(* IEC 61131-3 sources: LANTA/1.8QVPLC1.0/phase-calibration/codex-manual-v2-20260911, 4 files *)

(* ---- GVL_PhaseCal.st ---- *)
{attribute 'qualified_only'}
VAR_GLOBAL
    (* Commands: non-retained. Never FORCE these or axis commands. *)
    xStart : BOOL;
    xAbort : BOOL;
    xReset : BOOL;
    (* Commissioning interlock: confirm aligned reads with the actual protocol first.
       recSize>=16 alone is NOT a frame/header/checksum verification. *)
    xRxAlignmentConfirmed : BOOL := FALSE;
    lrCurrentPhaseDeg : LREAL := 0;
    iPhaseDirection : INT := 0; (* unknown=0, CCW=+1, CW=-1 *)
    (* Manual configuration. HPBW is the FULL -3 dB width in degrees. *)
    lrBeamAzDeg : LREAL := 0; (* required *)
    lrBeamElDeg : LREAL := 0; (* required *)
    lrScanFraction : LREAL := 0.2;
    lrTargetVolt : LREAL := 1.0; (* at 0.2 HPBW, independent of scan fraction *)
    lrCurrentGainAz : LREAL := 1;
    lrCurrentGainEl : LREAL := 1;
    iGainUnit : INT := 0; (* 0=linear voltage multiplier; 1=20*log10 multiplier dB *)
    iGainOrder : INT := 0; (* required: 1=gains before common rotation; 2=after *)
    lrGainMin : LREAL := 0.01; (* limits in selected device gain units *)
    lrGainMax : LREAL := 100;
    lrLegTimeSec : LREAL := 1.1;
    lrSettleSec : LREAL := 0.6; (* total dwell, including delay/settling and collection *)
    lrRxDelaySec : LREAL := 0.15; (* measured upper bound of receiver/filter delay *)
    lrStableSec : LREAL := 0.10;
    lrSampleIntervalSec : LREAL := 0.02;
    lrPositionToleranceDeg : LREAL := 0.002; (* mechanical per-axis *)
    lrMaxAxisOffsetDeg : LREAL := 0.1; (* commissioning ceiling; explicitly review if changed *)
    lrMaxVelocityDegSec : LREAL := 0; (* required mechanical per-axis limit *)
    lrMaxAccelerationDegSec2 : LREAL := 0; (* required mechanical per-axis limit *)
    lrMinCosEl : LREAL := 0.1; (* reject near zenith *)
    lrMaxOrthErrorDeg : LREAL := 3;
    lrMinEbN0 : LREAL := 29; (* legacy compatibility; no new EbN0 gate *)

    xGainValid : BOOL;
    lrGainFactorAz, lrGainFactorEl : LREAL;
    lrSuggestedGainAz, lrSuggestedGainEl : LREAL;
    lrSensitivityAz, lrSensitivityEl : LREAL; (* V/degree after proposed rotation, before new gain *)
    lrTargetSlopeAz, lrTargetSlopeEl : LREAL;
    lrPlannedTimeSec, lrCenterElevationDeg, lrProjectionCos : LREAL;
    lrPlannedAzOffsetDeg, lrPlannedElOffsetDeg : LREAL;
    lrCenterUa, lrCenterUe : LREAL; (* fitted center voltages, NOT proven electronic zero *)
    udiCenterSamples, udiElSamples, udiAzSamples, udiReturnSamples : UDINT;

    xReady, xBusy, xDone, xFault, xAborted : BOOL;
    xFitValid, xSuggestedValid : BOOL;
    uiError, uiFitError, uiState : UINT;
    udiSamples : UDINT;
    lrAzBias, lrElBias, lrRxAgeSec : LREAL;
    lrResponseAngleDeg, lrCorrectionDeg, lrSuggestedDeg : LREAL;
    lrCandidatePlusDeg, lrCandidateMinusDeg : LREAL;
    lrOrthErrorDeg, lrResidualAz, lrResidualEl : LREAL;
    lrKaa, lrKae, lrKea, lrKee : LREAL;

    (* SerialCom single writer; Canopen single reader. Even/odd sequence lock.
       Positions are PLC feedback at receive time, not sender timestamps. *)
    udiRxSeq : UDINT;
    uiReadSize, uiSerialError : UINT;
    udiReadCount, udiShortReadCount : UDINT;
    lrRxUa, lrRxUe, lrRxEbN0, lrRxAz, lrRxEl : LREAL;
    xRxLock : BOOL;
END_VAR

(* ---- FB_PhaseFit.st ---- *)
FUNCTION_BLOCK FB_PhaseFit
(* Offline candidate. Feed ONE coherent, validated sample per xSample pulse.
   Coordinates: positive Az=right, positive El=up. Desired response is -I.
   eAz/eEl must already have consistent signed engineering units.
   Do not subtract 2.5 from the existing signed serial values without protocol proof. *)
VAR_INPUT
    xReset : BOOL;
    xSample : BOOL;
    xFinish : BOOL;
    lrAz : LREAL;
    lrEl : LREAL;
    lrUa : LREAL;
    lrUe : LREAL;
    lrCurrentPhaseDeg : LREAL;
    (* +1: increasing hardware phase rotates measured response CCW; -1: CW; 0: unknown *)
    iPhaseDirection : INT;
END_VAR
VAR_OUTPUT
    xFitValid : BOOL;
    xSuggestedValid : BOOL;
    uiError : UINT;
    udiSamples : UDINT;
    lrKaa, lrKae, lrKea, lrKee : LREAL;
    lrInterceptAz, lrInterceptEl : LREAL;
    lrResponseAngleDeg : LREAL;
    lrCorrectionDeg, lrSuggestedDeg : LREAL;
    lrCandidatePlusDeg, lrCandidateMinusDeg : LREAL;
    lrOrthErrorDeg : LREAL;
    lrResidualAz, lrResidualEl : LREAL;
    lrCrossAz, lrCrossEl : LREAL;
END_VAR
VAR
    sx, sy, su, sv, sxx, syy, sxy, sxu, syu, sxv, syv, suu, svv : LREAL;
    n, xx, yy, xy, xu, yu, xv, yv, uu, vv, det : LREAL;
    ga, lrElGain, dot, a, b, phi, pi, base, sse : LREAL;
    finishOld : BOOL;
END_VAR

pi := 3.141592653589793;
IF xReset THEN
    sx:=0; sy:=0; su:=0; sv:=0; sxx:=0; syy:=0; sxy:=0;
    sxu:=0; syu:=0; sxv:=0; syv:=0; suu:=0; svv:=0;
    udiSamples:=0; uiError:=0; xFitValid:=FALSE; xSuggestedValid:=FALSE;
    lrKaa:=0; lrKae:=0; lrKea:=0; lrKee:=0;
    lrInterceptAz:=0; lrInterceptEl:=0; lrResponseAngleDeg:=0;
    lrCorrectionDeg:=0; lrSuggestedDeg:=0;
    lrCandidatePlusDeg:=0; lrCandidateMinusDeg:=0;
    lrOrthErrorDeg:=0; lrResidualAz:=0; lrResidualEl:=0;
    lrCrossAz:=0; lrCrossEl:=0;
ELSIF xSample AND NOT xFinish THEN
    IF udiSamples < 100000 THEN
        udiSamples:=udiSamples+1;
        sx:=sx+lrAz; sy:=sy+lrEl; su:=su+lrUa; sv:=sv+lrUe;
        sxx:=sxx+lrAz*lrAz; syy:=syy+lrEl*lrEl; sxy:=sxy+lrAz*lrEl;
        sxu:=sxu+lrAz*lrUa; syu:=syu+lrEl*lrUa;
        sxv:=sxv+lrAz*lrUe; syv:=syv+lrEl*lrUe;
        suu:=suu+lrUa*lrUa; svv:=svv+lrUe*lrUe;
    ELSE
        uiError:=1;
    END_IF;
END_IF;

IF xFinish AND NOT finishOld AND NOT xReset THEN
    xFitValid:=FALSE; xSuggestedValid:=FALSE;
    IF udiSamples < 30 OR uiError <> 0 THEN
        uiError:=2;
    ELSE
        n:=UDINT_TO_LREAL(udiSamples);
        xx:=sxx-sx*sx/n; yy:=syy-sy*sy/n; xy:=sxy-sx*sy/n;
        xu:=sxu-sx*su/n; yu:=syu-sy*su/n;
        xv:=sxv-sx*sv/n; yv:=syv-sy*sv/n;
        uu:=suu-su*su/n; vv:=svv-sv*sv/n;
        det:=xx*yy-xy*xy;
        IF xx <= 1E-12 OR yy <= 1E-12 OR det <= 0.01*xx*yy THEN
            uiError:=3; (* insufficient two-axis excitation *)
        ELSE
            lrKaa:=(xu*yy-yu*xy)/det;
            lrKae:=(yu*xx-xu*xy)/det;
            lrKea:=(xv*yy-yv*xy)/det;
            lrKee:=(yv*xx-xv*xy)/det;
            lrInterceptAz:=(su-lrKaa*sx-lrKae*sy)/n;
            lrInterceptEl:=(sv-lrKea*sx-lrKee*sy)/n;
            ga:=SQRT(lrKaa*lrKaa+lrKea*lrKea);
            lrElGain:=SQRT(lrKae*lrKae+lrKee*lrKee);
            sse:=MAX(0.0,uu-lrKaa*xu-lrKae*yu);
            lrResidualAz:=SQRT(sse/n);
            sse:=MAX(0.0,vv-lrKea*xv-lrKee*yv);
            lrResidualEl:=SQRT(sse/n);
            IF ga < 1E-6 OR lrElGain < 1E-6 OR (uu+vv) < 1E-10 THEN
                uiError:=4; (* no usable response *)
            ELSIF (lrKaa*lrKee-lrKae*lrKea) <= 0 THEN
                uiError:=5; (* reflection/polarity mismatch; common rotation cannot fix *)
            ELSE
                dot:=(lrKaa*lrKae+lrKea*lrKee)/(ga*lrElGain);
                dot:=LIMIT(-1.0,dot,1.0);
                lrOrthErrorDeg:=ABS(90.0-ACOS(dot)*180.0/pi);
                (* Normalize columns to prevent unequal axis gains dominating angle.
                   For M=R(phi)*diag(-ga,-lrElGain), a=2*cos(phi), b=2*sin(phi). *)
                a:=-lrKaa/ga-lrKee/lrElGain;
                b:=-lrKea/ga+lrKae/lrElGain;
                IF ABS(a)+ABS(b)<1E-9 THEN
                    uiError:=6;
                ELSE
                    IF ABS(a)<1E-12 THEN
                        IF b>=0 THEN phi:=pi/2; ELSE phi:=-pi/2; END_IF;
                    ELSE
                        phi:=ATAN(b/a);
                        IF a<0 THEN
                            IF b>=0 THEN phi:=phi+pi; ELSE phi:=phi-pi; END_IF;
                        END_IF;
                    END_IF;
                    lrResponseAngleDeg:=phi*180.0/pi;
                    (* Finite diagnostic ratio; 1E6 means a vanishing main channel. *)
                    lrCrossAz:=ABS(lrKea)/MAX(ABS(lrKaa),ga*1E-6);
                    lrCrossEl:=ABS(lrKae)/MAX(ABS(lrKee),lrElGain*1E-6);
                    (* Orthogonality is diagnostic only during commissioning.
                       xFitValid means rotation-estimate checks passed, NOT full calibration.
                       Keep residual rejection and all other validity checks unchanged. *)
                    IF (lrResidualAz*lrResidualAz+lrResidualEl*lrResidualEl)*n > 0.1*(uu+vv) THEN
                        uiError:=7; (* residual too large; correction rejected *)
                    ELSIF lrCurrentPhaseDeg<0 OR lrCurrentPhaseDeg>360 THEN
                        uiError:=8;
                    ELSE
                        xFitValid:=TRUE;
                        base:=lrCurrentPhaseDeg;
                        lrCandidatePlusDeg:=base+lrResponseAngleDeg;
                        lrCandidateMinusDeg:=base-lrResponseAngleDeg;
                        IF lrCandidatePlusDeg<0 THEN lrCandidatePlusDeg:=lrCandidatePlusDeg+360; END_IF;
                        IF lrCandidatePlusDeg>=360 THEN lrCandidatePlusDeg:=lrCandidatePlusDeg-360; END_IF;
                        IF lrCandidateMinusDeg<0 THEN lrCandidateMinusDeg:=lrCandidateMinusDeg+360; END_IF;
                        IF lrCandidateMinusDeg>=360 THEN lrCandidateMinusDeg:=lrCandidateMinusDeg-360; END_IF;
                        IF iPhaseDirection=1 OR iPhaseDirection=-1 THEN
                            lrCorrectionDeg:=-lrResponseAngleDeg/INT_TO_LREAL(iPhaseDirection);
                            lrSuggestedDeg:=base+lrCorrectionDeg;
                            IF lrSuggestedDeg<0 THEN lrSuggestedDeg:=lrSuggestedDeg+360; END_IF;
                            IF lrSuggestedDeg>=360 THEN lrSuggestedDeg:=lrSuggestedDeg-360; END_IF;
                            xSuggestedValid:=TRUE;
                        END_IF;
                    END_IF;
                END_IF;
            END_IF;
        END_IF;
    END_IF;
END_IF;
finishOld:=xFinish AND NOT xReset;
END_FUNCTION_BLOCK

(* ---- FB_PhaseTriangle.st ---- *)
FUNCTION_BLOCK FB_PhaseTriangle
(* Pure offset generator. Does NOT write axis commands or change operating modes.
   Caller supplies elapsed seconds and motion permission; xStart is rising-edge.
   xAbort returns offsets smoothly while permission remains valid.
   Permission loss holds offsets and sets xFault: existing axis safety owns stopping.
   Release a held offset only after the caller has safely transferred command ownership. *)
VAR_INPUT
    xStart, xAbort, xPermit : BOOL;
    xResetHeld : BOOL;
    lrDtSec : LREAL;
    lrAzAmplitudeDeg, lrElAmplitudeDeg : LREAL;
    lrLegTimeSec : LREAL := 1.1;
    lrSettleSec : LREAL := 0.6;
END_VAR
VAR_OUTPUT
    xBusy, xDone, xAborted, xFault : BOOL;
    uiState : UINT;
    lrAzBias, lrElBias : LREAL;
    xCollect : BOOL;
END_VAR
VAR
    startOld : BOOL;
    elapsed, leg, settle, azAmplitude, elAmplitude, u, blend : LREAL;
    fromAz, fromEl, toAz, toEl : LREAL;
END_VAR

xCollect:=FALSE;
IF xResetHeld AND NOT xPermit AND uiState=900 THEN
    uiState:=0; xBusy:=FALSE; xFault:=FALSE;
    lrAzBias:=0; lrElBias:=0;
END_IF;
IF xStart AND NOT startOld AND NOT xBusy AND uiState<>900 THEN
    xDone:=FALSE; xAborted:=FALSE; xFault:=FALSE;
    (* Caller validates projected amplitudes and mechanical motion limits. *)
    IF NOT xPermit OR lrAzAmplitudeDeg<=0 OR lrElAmplitudeDeg<=0 OR
       lrLegTimeSec<0.2 OR lrSettleSec<0.1 OR lrSettleSec>30 THEN
        xFault:=TRUE;
    ELSE
        azAmplitude:=lrAzAmplitudeDeg; elAmplitude:=lrElAmplitudeDeg;
        leg:=lrLegTimeSec; settle:=lrSettleSec;
        elapsed:=0; lrAzBias:=0; lrElBias:=0;
        uiState:=10; xBusy:=TRUE;
    END_IF;
END_IF;
startOld:=xStart;

IF xBusy AND uiState<>900 THEN
    IF NOT xPermit OR lrDtSec<=0 OR lrDtSec>0.1 THEN
        xFault:=TRUE; uiState:=900;
    ELSE
        IF xAbort AND uiState<>800 THEN
            fromAz:=lrAzBias; fromEl:=lrElBias;
            toAz:=0; toEl:=0; elapsed:=0;
            xAborted:=TRUE; uiState:=800;
        END_IF;
        elapsed:=elapsed+lrDtSec;
        CASE uiState OF
            10,30,50,70:
                xCollect:=TRUE; (* caller still gates new-frame, quality, position settling *)
                IF elapsed>=settle THEN
                    elapsed:=0; fromAz:=lrAzBias; fromEl:=lrElBias;
                    CASE uiState OF
                        10: toAz:=0; toEl:=elAmplitude; uiState:=20;
                        30: toAz:=azAmplitude; toEl:=0; uiState:=40;
                        50: toAz:=0; toEl:=0; uiState:=60;
                        70: xBusy:=FALSE; xDone:=TRUE; uiState:=0;
                    END_CASE;
                END_IF;
            20,40,60,800:
                u:=LIMIT(0.0,elapsed/leg,1.0);
                blend:=u*u*u*(10.0+u*(-15.0+6.0*u));
                lrAzBias:=fromAz+(toAz-fromAz)*blend;
                lrElBias:=fromEl+(toEl-fromEl)*blend;
                xCollect:=FALSE; (* stationary samples only *)
                IF u>=1 THEN
                    elapsed:=0;
                    IF uiState=800 THEN
                        xBusy:=FALSE; uiState:=0;
                    ELSE
                        uiState:=uiState+10;
                    END_IF;
                END_IF;
        END_CASE;
    END_IF;
END_IF;
END_FUNCTION_BLOCK

(* ---- PRG_PhaseCalibration.st ---- *)
PROGRAM PRG_PhaseCalibration
(* Called ONLY at the end of SecurityCheck, once per Canopen 10 ms cycle.
   Fixed position mode only. No writes to modes, enables, tracking or persistence.
   Loss of ownership gives command control back to the existing program immediately.
   This is not an emergency-stop/safety function. *)
VAR
    path : FB_PhaseTriangle;
    fit : FB_PhaseFit;
    startOld, startPulse, accepted, permit, ownership : BOOL;
    sample, finish, newRx, rxLock, doneOld, abortRun : BOOL;
    seq, lastSeq : UDINT;
    age : LREAL := 999;
    sampleTime : LREAL;
    ua, ue, eb, az, el, centerAz, centerEl : LREAL;
    baseAz, baseEl, phase : LREAL;
    direction : INT;
    beamAz, beamEl, fraction, targetV, cosEl, azAmplitude, elAmplitude : LREAL;
    gainAz, gainEl, currentGainAz, currentGainEl, gainMin, gainMax : LREAL;
    gainUnit, gainOrder : INT;
    legTime, dwellTime, rxDelay, stableTime, interval, tolerance, orthLimit : LREAL;
    stableElapsed, normUa, normUe, slopeAz, slopeEl, factorAz, factorEl : LREAL;
    previousState : UINT;
    centerCount, elCount, azCount, returnCount : UDINT;
    geometryOK, configOK : BOOL;
END_VAR

startPulse:=GVL_PhaseCal.xStart AND NOT startOld;
startOld:=GVL_PhaseCal.xStart;
accepted:=FALSE; sample:=FALSE; newRx:=FALSE;
age:=MIN(age+0.01,999.0);
sampleTime:=MIN(sampleTime+0.01,1.0);
seq:=GVL_PhaseCal.udiRxSeq;
IF seq<>lastSeq AND seq MOD 2=0 THEN
    ua:=GVL_PhaseCal.lrRxUa; ue:=GVL_PhaseCal.lrRxUe;
    eb:=GVL_PhaseCal.lrRxEbN0;
    az:=GVL_PhaseCal.lrRxAz; el:=GVL_PhaseCal.lrRxEl;
    rxLock:=GVL_PhaseCal.xRxLock;
    IF seq=GVL_PhaseCal.udiRxSeq THEN
        lastSeq:=seq; age:=0; newRx:=TRUE;
    END_IF;
END_IF;

ownership:=NOT GVL.bLocalCtrl AND GVL.Axis1Remote.iMode=2 AND
    GVL.Axis2Remote.iMode=2 AND NOT GVL.bStartTrack AND
    NOT GVL.bStartLocalAutoTrack AND NOT Modbus_Slave.bStartTrackAcu AND
    NOT Modbus_Slave.bSearch AND NOT SecurityCheck.bScanRun AND
    ABS(SecurityCheck.aztest)<0.00001 AND ABS(SecurityCheck.eltest)<0.00001;
permit:=ownership AND GVL.Axis1Status.bServo_Enable AND
    GVL.Axis2Status.bServo_Enable AND NOT GVL.Axis1Status.Error AND
    NOT GVL.Axis2Status.Error AND NOT GVL.Axis1Status.ErrorStop AND
    NOT GVL.Axis2Status.ErrorStop AND GVL.eAzErrorcode=0 AND GVL.eElErrorcode=0 AND
    NOT SecurityCheck.bPrelimit_1 AND NOT SecurityCheck.bPrelimit_2 AND
    NOT SecurityCheck.bFinallimit_1 AND NOT SecurityCheck.bFinallimit_2;
IF path.xBusy THEN
    (* Never mask a changed ACU target by holding the old calibration center. *)
    permit:=permit AND ABS(REAL_TO_LREAL(Modbus_Slave.rPosCmd_2)-baseAz)<0.00001 AND
        ABS(REAL_TO_LREAL(Modbus_Slave.rPosCmd_1)-baseEl)<0.00001;
END_IF;
(* Signal quality and initial pointing are assessed manually by the operator.
   Keep new-receive sampling; never manufacture samples from stale values. *)
GVL_PhaseCal.xReady:=permit AND
    NOT path.xBusy AND NOT GVL_PhaseCal.xFault AND NOT GVL_PhaseCal.xAbort AND
    ABS(REAL_TO_LREAL(Modbus_Slave.rPosCmd_2))<274.8 AND
    Modbus_Slave.rPosCmd_1>93.2 AND Modbus_Slave.rPosCmd_1<179.8;

IF GVL_PhaseCal.xReset AND NOT path.xBusy THEN
    GVL_PhaseCal.xFault:=FALSE; GVL_PhaseCal.uiError:=0;
END_IF;
IF startPulse AND NOT path.xBusy THEN
    GVL_PhaseCal.xGainValid:=FALSE;
    GVL_PhaseCal.lrGainFactorAz:=0; GVL_PhaseCal.lrGainFactorEl:=0;
    GVL_PhaseCal.lrSuggestedGainAz:=0; GVL_PhaseCal.lrSuggestedGainEl:=0;
    beamAz:=GVL_PhaseCal.lrBeamAzDeg; beamEl:=GVL_PhaseCal.lrBeamElDeg;
    fraction:=GVL_PhaseCal.lrScanFraction; targetV:=GVL_PhaseCal.lrTargetVolt;
    legTime:=GVL_PhaseCal.lrLegTimeSec; dwellTime:=GVL_PhaseCal.lrSettleSec;
    rxDelay:=GVL_PhaseCal.lrRxDelaySec; stableTime:=GVL_PhaseCal.lrStableSec;
    interval:=GVL_PhaseCal.lrSampleIntervalSec; tolerance:=GVL_PhaseCal.lrPositionToleranceDeg;
    orthLimit:=GVL_PhaseCal.lrMaxOrthErrorDeg;
    currentGainAz:=GVL_PhaseCal.lrCurrentGainAz; currentGainEl:=GVL_PhaseCal.lrCurrentGainEl;
    gainUnit:=GVL_PhaseCal.iGainUnit; gainOrder:=GVL_PhaseCal.iGainOrder;
    gainMin:=GVL_PhaseCal.lrGainMin; gainMax:=GVL_PhaseCal.lrGainMax;
    GVL_PhaseCal.lrCenterElevationDeg:=REAL_TO_LREAL(Modbus_Slave.rPosCmd_1)-90;
    cosEl:=COS(GVL_PhaseCal.lrCenterElevationDeg*3.141592653589793/180);
    geometryOK:=beamAz>0 AND beamEl>0 AND beamAz<=10 AND beamEl<=10 AND
        fraction>=0.05 AND fraction<=0.2 AND GVL_PhaseCal.lrMinCosEl>=0.05 AND
        GVL_PhaseCal.lrMinCosEl<=1 AND cosEl>=GVL_PhaseCal.lrMinCosEl;
    azAmplitude:=0; elAmplitude:=0;
    IF geometryOK THEN azAmplitude:=fraction*beamAz/cosEl; elAmplitude:=fraction*beamEl; END_IF;
    gainAz:=0; gainEl:=0;
    IF gainUnit=0 THEN gainAz:=currentGainAz; gainEl:=currentGainEl;
    ELSIF gainUnit=1 AND ABS(currentGainAz)<=120 AND ABS(currentGainEl)<=120 THEN
        gainAz:=EXP(currentGainAz*LN(10.0)/20); gainEl:=EXP(currentGainEl*LN(10.0)/20);
    END_IF;
    configOK:=geometryOK AND gainAz>=1E-6 AND gainEl>=1E-6 AND
        (gainOrder=1 OR gainOrder=2) AND gainMin<gainMax AND
        currentGainAz>=gainMin AND currentGainAz<=gainMax AND
        currentGainEl>=gainMin AND currentGainEl<=gainMax AND
        targetV>0 AND targetV<=4 AND legTime>=0.2 AND legTime<=60 AND
        dwellTime>=0.1 AND dwellTime<=30 AND rxDelay>=0 AND stableTime>=0.05 AND
        interval>=0.01 AND interval<=0.2 AND dwellTime>rxDelay+stableTime+5*interval AND
        tolerance>0 AND tolerance<0.1*MIN(azAmplitude,elAmplitude) AND
        orthLimit>0 AND orthLimit<=10 AND
        GVL_PhaseCal.lrMaxAxisOffsetDeg>0 AND GVL_PhaseCal.lrMaxAxisOffsetDeg<=1 AND
        MAX(azAmplitude,elAmplitude)<=GVL_PhaseCal.lrMaxAxisOffsetDeg AND
        ABS(REAL_TO_LREAL(Modbus_Slave.rPosCmd_2)-azAmplitude)<274.8 AND
        REAL_TO_LREAL(Modbus_Slave.rPosCmd_1)+elAmplitude<179.8 AND
        NOT GVL_PhaseCal.xReset;
    IF legTime>=0.2 THEN
        configOK:=configOK AND 1.875*MAX(azAmplitude,elAmplitude)/legTime<=GVL_PhaseCal.lrMaxVelocityDegSec AND
            5.774*MAX(azAmplitude,elAmplitude)/(legTime*legTime)<=GVL_PhaseCal.lrMaxAccelerationDegSec2;
    END_IF;
    GVL_PhaseCal.lrPlannedTimeSec:=3*legTime+4*dwellTime;
    GVL_PhaseCal.lrProjectionCos:=cosEl;
    GVL_PhaseCal.lrPlannedAzOffsetDeg:=azAmplitude; GVL_PhaseCal.lrPlannedElOffsetDeg:=elAmplitude;
    GVL_PhaseCal.xDone:=FALSE;
    GVL_PhaseCal.xFitValid:=FALSE; GVL_PhaseCal.xSuggestedValid:=FALSE;
    IF NOT GVL_PhaseCal.xReady OR GVL_PhaseCal.lrCurrentPhaseDeg<0 OR
       GVL_PhaseCal.lrCurrentPhaseDeg>360 OR
       NOT configOK THEN
        GVL_PhaseCal.uiError:=10; GVL_PhaseCal.xFault:=TRUE;
    ELSE
        baseAz:=REAL_TO_LREAL(Modbus_Slave.rPosCmd_2);
        baseEl:=REAL_TO_LREAL(Modbus_Slave.rPosCmd_1);
        centerAz:=-baseAz; centerEl:=baseEl-90;
        phase:=GVL_PhaseCal.lrCurrentPhaseDeg;
        direction:=GVL_PhaseCal.iPhaseDirection;
        accepted:=TRUE; sampleTime:=0; stableElapsed:=0;
        centerCount:=0; elCount:=0; azCount:=0; returnCount:=0;
        GVL_PhaseCal.uiError:=0; GVL_PhaseCal.xFault:=FALSE;
    END_IF;
END_IF;

abortRun:=GVL_PhaseCal.xAbort;
IF path.xBusy AND path.uiState<>800 AND path.uiState<>900 THEN
    IF ABS(-REAL_TO_LREAL(GVL.rFctPosReal_2)-centerAz-path.lrAzBias)>0.1 OR
       ABS(REAL_TO_LREAL(GVL.rFctPosReal_1)-90-centerEl-path.lrElBias)>0.1 THEN
        abortRun:=TRUE; GVL_PhaseCal.uiError:=21; GVL_PhaseCal.xFault:=TRUE;
    END_IF;
END_IF;
path(xStart:=accepted, xAbort:=abortRun, xPermit:=permit,
    xResetHeld:=GVL_PhaseCal.xReset AND NOT GVL.Axis1Status.bServo_Enable AND
        NOT GVL.Axis2Status.bServo_Enable,
    lrDtSec:=0.01, lrAzAmplitudeDeg:=azAmplitude, lrElAmplitudeDeg:=elAmplitude,
    lrLegTimeSec:=legTime, lrSettleSec:=dwellTime);
IF path.xFault THEN
    GVL_PhaseCal.xFault:=TRUE; GVL_PhaseCal.uiError:=22;
END_IF;
IF path.xBusy AND permit AND path.uiState<>900 THEN
    (* Same signs as existing eltest/aztest target offsets. *)
    GVL.Axis1Remote.rPosCmd:=LREAL_TO_REAL(baseEl+path.lrElBias);
    GVL.Axis2Remote.rPosCmd:=LREAL_TO_REAL(baseAz-path.lrAzBias);
END_IF;
(* Wait continuously at the commanded vertex; then allow receiver history to flush.
   Positions are mechanical feedback. No moving samples and no synthetic new frames. *)
IF path.uiState<>previousState THEN stableElapsed:=0; END_IF;
previousState:=path.uiState;
IF path.xBusy AND path.xCollect AND
   ABS(-REAL_TO_LREAL(GVL.rFctPosReal_2)-centerAz-path.lrAzBias)<=tolerance AND
   ABS(REAL_TO_LREAL(GVL.rFctPosReal_1)-90-centerEl-path.lrElBias)<=tolerance THEN
    stableElapsed:=stableElapsed+0.01;
ELSE stableElapsed:=0;
END_IF;
IF path.xBusy AND path.xCollect AND stableElapsed>=rxDelay+stableTime AND
   newRx AND sampleTime>=interval AND NOT GVL_PhaseCal.xFault AND NOT path.xAborted AND
   ABS(az-centerAz-path.lrAzBias)<=tolerance AND ABS(el-centerEl-path.lrElBias)<=tolerance THEN
    sample:=TRUE; sampleTime:=0;
    CASE path.uiState OF
        10: centerCount:=centerCount+1;
        30: elCount:=elCount+1;
        50: azCount:=azCount+1;
        70: returnCount:=returnCount+1;
    END_CASE;
END_IF;
finish:=path.xDone AND NOT doneOld AND NOT GVL_PhaseCal.xFault;
IF finish AND (ABS(-REAL_TO_LREAL(GVL.rFctPosReal_2)-centerAz)>tolerance OR
              ABS(REAL_TO_LREAL(GVL.rFctPosReal_1)-90-centerEl)>tolerance) THEN
    finish:=FALSE; GVL_PhaseCal.xFault:=TRUE; GVL_PhaseCal.uiError:=31;
END_IF;
IF finish AND (centerCount<5 OR elCount<5 OR azCount<5 OR returnCount<5) THEN
    finish:=FALSE; GVL_PhaseCal.xFault:=TRUE; GVL_PhaseCal.uiError:=32;
END_IF;
doneOld:=path.xDone;
normUa:=ua; normUe:=ue;
(* Known post-rotation gains must be removed before fitting a common rotation. *)
IF gainOrder=2 AND gainAz>0 AND gainEl>0 THEN normUa:=ua/gainAz; normUe:=ue/gainEl; END_IF;
fit(xReset:=accepted, xSample:=sample, xFinish:=finish,
    lrAz:=(az-centerAz)*cosEl, lrEl:=el-centerEl, lrUa:=normUa, lrUe:=normUe,
    lrCurrentPhaseDeg:=phase, iPhaseDirection:=direction);
IF finish THEN
    GVL_PhaseCal.xDone:=TRUE;
    GVL_PhaseCal.xFitValid:=fit.xFitValid;
    GVL_PhaseCal.xSuggestedValid:=fit.xSuggestedValid;
    IF NOT fit.xFitValid THEN
        GVL_PhaseCal.xFault:=TRUE; GVL_PhaseCal.uiError:=30;
    END_IF;
END_IF;
IF finish AND fit.xFitValid THEN
    slopeAz:=SQRT(fit.lrKaa*fit.lrKaa+fit.lrKea*fit.lrKea);
    slopeEl:=SQRT(fit.lrKae*fit.lrKae+fit.lrKee*fit.lrKee);
    GVL_PhaseCal.lrCenterUa:=fit.lrInterceptAz; GVL_PhaseCal.lrCenterUe:=fit.lrInterceptEl;
    IF gainOrder=2 THEN
        slopeAz:=slopeAz*gainAz; slopeEl:=slopeEl*gainEl;
        GVL_PhaseCal.lrCenterUa:=fit.lrInterceptAz*gainAz;
        GVL_PhaseCal.lrCenterUe:=fit.lrInterceptEl*gainEl;
    END_IF;
    GVL_PhaseCal.lrSensitivityAz:=slopeAz; GVL_PhaseCal.lrSensitivityEl:=slopeEl;
    GVL_PhaseCal.lrTargetSlopeAz:=targetV/(0.2*beamAz);
    GVL_PhaseCal.lrTargetSlopeEl:=targetV/(0.2*beamEl);
    IF slopeAz>1E-6 AND slopeEl>1E-6 AND fit.lrOrthErrorDeg<=orthLimit THEN
        factorAz:=GVL_PhaseCal.lrTargetSlopeAz/slopeAz;
        factorEl:=GVL_PhaseCal.lrTargetSlopeEl/slopeEl;
        GVL_PhaseCal.lrGainFactorAz:=factorAz; GVL_PhaseCal.lrGainFactorEl:=factorEl;
        IF gainUnit=0 THEN
            GVL_PhaseCal.lrSuggestedGainAz:=currentGainAz*factorAz;
            GVL_PhaseCal.lrSuggestedGainEl:=currentGainEl*factorEl;
        ELSE
            GVL_PhaseCal.lrSuggestedGainAz:=currentGainAz+20*LN(factorAz)/LN(10.0);
            GVL_PhaseCal.lrSuggestedGainEl:=currentGainEl+20*LN(factorEl)/LN(10.0);
        END_IF;
        GVL_PhaseCal.xGainValid:=fit.xSuggestedValid AND
            GVL_PhaseCal.lrSuggestedGainAz>=gainMin AND GVL_PhaseCal.lrSuggestedGainAz<=gainMax AND
            GVL_PhaseCal.lrSuggestedGainEl>=gainMin AND GVL_PhaseCal.lrSuggestedGainEl<=gainMax;
    END_IF;
END_IF;
GVL_PhaseCal.udiCenterSamples:=centerCount; GVL_PhaseCal.udiElSamples:=elCount;
GVL_PhaseCal.udiAzSamples:=azCount; GVL_PhaseCal.udiReturnSamples:=returnCount;
GVL_PhaseCal.xBusy:=path.xBusy; GVL_PhaseCal.xAborted:=path.xAborted;
GVL_PhaseCal.uiState:=path.uiState; GVL_PhaseCal.uiFitError:=fit.uiError;
GVL_PhaseCal.lrAzBias:=path.lrAzBias; GVL_PhaseCal.lrElBias:=path.lrElBias;
GVL_PhaseCal.lrRxAgeSec:=age; GVL_PhaseCal.udiSamples:=fit.udiSamples;
GVL_PhaseCal.lrResponseAngleDeg:=fit.lrResponseAngleDeg;
GVL_PhaseCal.lrCorrectionDeg:=fit.lrCorrectionDeg;
GVL_PhaseCal.lrSuggestedDeg:=fit.lrSuggestedDeg;
GVL_PhaseCal.lrCandidatePlusDeg:=fit.lrCandidatePlusDeg;
GVL_PhaseCal.lrCandidateMinusDeg:=fit.lrCandidateMinusDeg;
GVL_PhaseCal.lrOrthErrorDeg:=fit.lrOrthErrorDeg;
GVL_PhaseCal.lrResidualAz:=fit.lrResidualAz; GVL_PhaseCal.lrResidualEl:=fit.lrResidualEl;
GVL_PhaseCal.lrKaa:=fit.lrKaa; GVL_PhaseCal.lrKae:=fit.lrKae;
GVL_PhaseCal.lrKea:=fit.lrKea; GVL_PhaseCal.lrKee:=fit.lrKee;
END_PROGRAM
